// TIA Portal project "SFC_Sep_Simples" (V16)

(* hardware
DEVICE "S71500/ET200MP station_1"  S7-1500 station
   slot 0: "Rail_0"  Rack  6ES7 590-1***0-0AA0
   slot 1: "PLC_1"  CPU 1512C-1 PN  6ES7 512-1CK00-0AB0  V2.8
      slot 3: "CPU display_1"  6ES7591-1AA00-0AA0
      slot 32768: "PROFINET interface_1"  X1
         slot 32769: "Port_1"  X1 P1
         slot 32770: "Port_2"  X1 P2
      slot 34817: "Virtual CP interface port_1"  Virtual CP interface port  Virtual CP interface port
*)

// ===== PLC "PLC_1"  CPU 1512C-1 PN =====

VAR_GLOBAL   // PLC tag table "Default tag table"
   "Count" AT %MW0 : Int;
END_VAR

VAR_GLOBAL   // PLC tag table "E_N_Controlaveis"
   "FIO_S3" AT %M5.3 : Bool;
   "FIO_S2" AT %M5.2 : Bool;
   "FIO_PA" AT %M5.1 : Bool;
   "FIO_PV" AT %M5.0 : Bool;
   "FIO_S4" AT %M5.5 : Bool;
   "FIO_AT_Fwd" AT %M5.6 : Bool;
   "FIOAT_Rev" AT %M5.7 : Bool;
END_VAR

VAR_GLOBAL   // PLC tag table "Saidas"
   "FIO_Atuador" AT %M10.0 : Bool;
   "FIO_Esteira1" AT %M10.1 : Bool;
   "FIO_Esteira2" AT %M10.2 : Bool;
   "FIO_Esteira4" AT %M10.4 : Bool;
   "FIO_Esteira3" AT %M10.3 : Bool;
END_VAR

// folder: DBs

DATA_BLOCK "Eventos"   // DB1
{ S7_Optimized_Access := 'TRUE' }
VERSION : 0.1
   VAR
      PV_Ev : Bool;
      PA_Ev : Bool;
      S2_On_Ev : Bool;
      S2_Off_Ev : Bool;
      S3_On_Ev : Bool;
      S3_Off_Ev : Bool;
      AT_Off_Ev : Bool;
      S4_Off_Ev : Bool;
      AT_On_Ev : Bool;
      E1_On_Ev : Bool;
      E1_Off_Ev : Bool;
      E2_On_Ev : Bool;
      E2_Off_Ev : Bool;
      E3_On_Ev : Bool;
      E3_Off_Ev : Bool;
   END_VAR
BEGIN
END_DATA_BLOCK

DATA_BLOCK "BitsAuxiliares"   // DB2
{ S7_Optimized_Access := 'TRUE' }
VERSION : 0.1
   VAR
      Aux1 : Bool;
      Aux2 : Bool;
      Cont : Int := 0;
   END_VAR
BEGIN
END_DATA_BLOCK

DATA_BLOCK "Sequencia_DB"   // DB6
{ S7_Optimized_Access := 'TRUE' }
VERSION : 0.1
// stored: InstanceOfName Sequencia
"Sequencia"
BEGIN
END_DATA_BLOCK

// folder: System blocks/Program resources

DATA_BLOCK "CT1"   // DB4
{ S7_Optimized_Access := 'TRUE' }
AUTHOR : Simatic
FAMILY : IEC
NAME : CNTR
VERSION : 1.0
// stored: InstanceOfName IEC_COUNTER
"IEC_COUNTER"
BEGIN
END_DATA_BLOCK

// folder: (top level)

ORGANIZATION_BLOCK "Main"   // OB1, LAD, ProgramCycle
TITLE = "Main Program Sweep (Cycle)"
{ S7_Optimized_Access := 'TRUE' }
VERSION : 0.1
   VAR_INPUT
      Initial_Call : Bool;   // Initial call of this OB
      Remanence : Bool;   // =True, if remanent data are available
   END_VAR
   VAR_TEMP   // added for the SCL form of the ladder/FBD networks
      _w1 : Bool;
      _w2 : Bool;
   END_VAR
BEGIN

REGION Network 1: Leituras De Borda
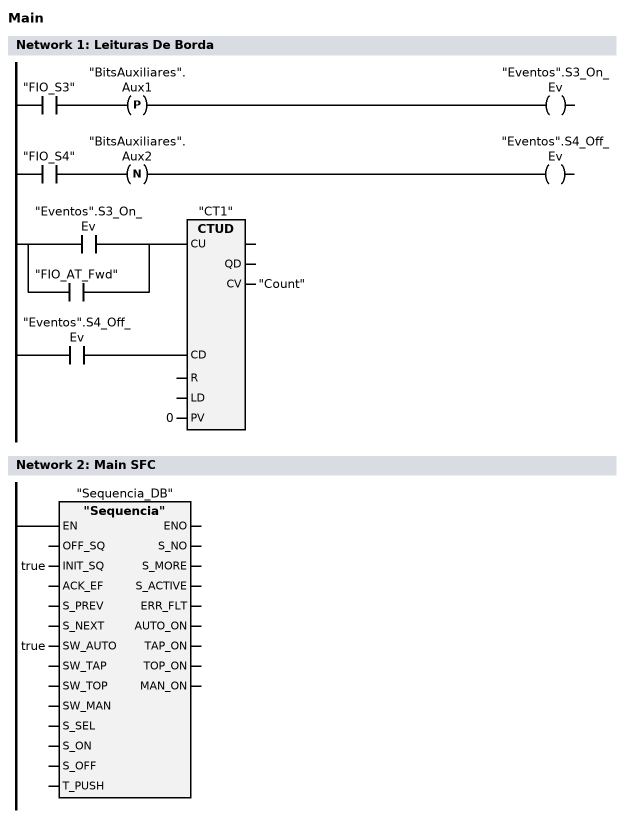
   #_w1 := "FIO_S3" AND NOT "BitsAuxiliares".Aux1;   // rising edge
   "BitsAuxiliares".Aux1 := "FIO_S3";
   "Eventos".S3_On_Ev := #_w1;
   #_w2 := NOT "FIO_S4" AND "BitsAuxiliares".Aux2;   // falling edge
   "BitsAuxiliares".Aux2 := "FIO_S4";
   "Eventos".S4_Off_Ev := #_w2;
   "CT1".CTUD(CU := "Eventos".S3_On_Ev OR "FIO_AT_Fwd", CD := "Eventos".S4_Off_Ev, PV := 0, CV => "Count");
END_REGION

REGION Network 2: Main SFC
   RUNG wire#powerrail
      "Sequencia_DB"(OFF_SQ :=, INIT_SQ := true, ACK_EF :=, S_PREV :=, S_NEXT :=, SW_AUTO := true, SW_TAP :=, SW_TOP :=, SW_MAN :=, S_SEL :=, S_ON :=, S_OFF :=, T_PUSH :=, S_NO =>, S_MORE =>, S_ACTIVE =>, ERR_FLT =>, AUTO_ON =>, TAP_ON =>, TOP_ON =>, MAN_ON =>)
   END_RUNG
   // the same network as SCL:
   "Sequencia_DB"(INIT_SQ := true, SW_AUTO := true);   // "Sequencia"
END_REGION
END_ORGANIZATION_BLOCK

// folder: FBs

FUNCTION_BLOCK "Sequencia"   // FB2, GRAPH_PLUS
{ S7_Optimized_Access := 'TRUE' }
VERSION : 0.1
   VAR_INPUT
      OFF_SQ : Bool := false;   // Turn sequence off
      INIT_SQ : Bool := false;   // Set sequence to initial state
      ACK_EF : Bool := false;   // Acknowledge all errors and faults
      S_PREV : Bool := false;   // Output previous step in parameter S_NO
      S_NEXT : Bool := false;   // Indicate next step in parameter S_NO
      SW_AUTO : Bool := false;   // Automatic mode
      SW_TAP : Bool := false;   // Semiautomatic/switch with transition
      SW_TOP : Bool := false;   // Semiautomatic/ignore transition
      SW_MAN : Bool := false;   // Manual mode
      S_SEL : Int := 0;   // Select step to be output to S_NO
      S_ON : Bool := false;   // Activate step indicated in S_NO
      S_OFF : Bool := false;   // Deactivate step indicated S_NO
      T_PUSH : Bool := false;   // Enable transition to switch in semi automatic mode
   END_VAR
   VAR_OUTPUT
      S_NO : Int := 0;   // Step number
      S_MORE : Bool := false;   // More steps are available and can be shown in S_NO
      S_ACTIVE : Bool := false;   // Step indicated in S_NO is active
      ERR_FLT : Bool := false;   // Interlock or supervision group error
      AUTO_ON : Bool := false;   // Automatic mode is active
      TAP_ON : Bool := false;   // Semiautomatic mode/step with transition enabled
      TOP_ON : Bool := false;   // Semiautomatic mode/ignore transition enabled
      MAN_ON : Bool := false;   // Manual mode is active
   END_VAR
   VAR
      HMI_INFO : Array[0..8] of UInt;
      IF_PAR : G7_IfParPlus_V6;
      RT_DATA : G7_RTDataPlus_V6;   // Internal data area
      Trans1 : G7_TransitionPlus_V6;   // Transition structure
      Trans2 : G7_TransitionPlus_V6;   // Transition structure
      Trans3 : G7_TransitionPlus_V6;   // Transition structure
      Trans4 : G7_TransitionPlus_V6;   // Transition structure
      Trans5 : G7_TransitionPlus_V6;   // Transition structure
      Trans6 : G7_TransitionPlus_V6;   // Transition structure
      Trans7 : G7_TransitionPlus_V6;   // Transition structure
      Trans8 : G7_TransitionPlus_V6;   // Transition structure
      Trans10 : G7_TransitionPlus_V6;   // Transition structure
      Trans12 : G7_TransitionPlus_V6;   // Transition structure
      Trans13 : G7_TransitionPlus_V6;   // Transition structure
      Trans14 : G7_TransitionPlus_V6;   // Transition structure
      Trans15 : G7_TransitionPlus_V6;   // Transition structure
      Trans16 : G7_TransitionPlus_V6;   // Transition structure
      Trans17 : G7_TransitionPlus_V6;   // Transition structure
      Step1 : G7_StepPlus_V6;   // Step structure
      Step2 : G7_StepPlus_V6;   // Step structure
      Step3 : G7_StepPlus_V6;   // Step structure
      Step4 : G7_StepPlus_V6;   // Step structure
      Step5 : G7_StepPlus_V6;   // Step structure
      Step6 : G7_StepPlus_V6;   // Step structure
      Step7 : G7_StepPlus_V6;   // Step structure
      Step9 : G7_StepPlus_V6;   // Step structure
      Step11 : G7_StepPlus_V6;   // Step structure
      Step12 : G7_StepPlus_V6;   // Step structure
      Step13 : G7_StepPlus_V6;   // Step structure
      SINI : Array[0..1] of USInt;
      LSTT : Array[0..14] of USInt;
      ATAJ : Array[0..14] of USInt;
      ATAB : Array[0..14] of USInt;
      PSTT : Array[0..14] of USInt;
      NSTT : Array[0..14] of USInt;
      ASSJ : Array[0..10] of USInt;
      ASSB : Array[0..10] of USInt;
      PTTS : Array[0..10] of USInt;
      NTTS : Array[0..10] of USInt;
      SW_SQTS : Array[0..10] of USInt;
      SWITCH : Array[0..3] of USInt;
      TVX : Array[0..7] of USInt;
      TTX : Array[0..7] of USInt;
      TSX : Array[0..1] of USInt;
      S00X : Array[0..1] of USInt;
      SOFFX : Array[0..1] of USInt;
      SONX : Array[0..1] of USInt;
      SAX : Array[0..1] of USInt;
      SERRX : Array[0..11] of USInt;
      SMX : Array[0..11] of USInt;
      S0X : Array[0..11] of USInt;
      S1X : Array[0..11] of USInt;
      IL_ALARM_INST : Diag_Alarm;
      SUP_ALARM_INST : Diag_Alarm;
      STEP_TIME_ALARM_INST : Diag_Alarm;
      IEC_TIMER_INST : IEC_TIMER;
      TRANSACTION_FLAG : Bool := false;
   END_VAR
   // SINI[0] := 2;
   // LSTT[0] := 255;
   // LSTT[1] := 255;
   // LSTT[2] := 255;
   // LSTT[3] := 255;
   // LSTT[4] := 255;
   // LSTT[5] := 255;
   // LSTT[6] := 255;
   // LSTT[7] := 255;
   // LSTT[8] := 4;
   // LSTT[9] := 255;
   // LSTT[11] := 5;
   // LSTT[12] := 7;
   // LSTT[13] := 255;
   // LSTT[14] := 8;
   // ATAJ[1] := 1;
   // ATAJ[2] := 2;
   // ATAJ[3] := 3;
   // ATAJ[4] := 4;
   // ATAJ[5] := 5;
   // ATAJ[6] := 6;
   // ATAJ[7] := 7;
   // ATAJ[8] := 8;
   // ATAJ[9] := 9;
   // ATAJ[10] := 10;
   // ATAJ[11] := 11;
   // ATAJ[12] := 12;
   // ATAJ[13] := 13;
   // ATAJ[14] := 14;
   // ATAB[1] := 1;
   // ATAB[2] := 2;
   // ATAB[3] := 12;
   // ATAB[4] := 3;
   // ATAB[5] := 5;
   // ATAB[6] := 7;
   // ATAB[7] := 6;
   // ATAB[8] := 8;
   // ATAB[9] := 9;
   // ATAB[10] := 10;
   // ATAB[11] := 4;
   // ATAB[12] := 11;
   // ATAB[13] := 13;
   // ATAB[14] := 14;
   // PSTT[1] := 1;
   // PSTT[2] := 2;
   // PSTT[3] := 3;
   // PSTT[4] := 3;
   // PSTT[5] := 4;
   // PSTT[6] := 10;
   // PSTT[7] := 10;
   // PSTT[8] := 7;
   // PSTT[9] := 8;
   // PSTT[10] := 9;
   // PSTT[11] := 3;
   // PSTT[12] := 3;
   // PSTT[13] := 5;
   // PSTT[14] := 6;
   // NSTT[0] := 1;
   // NSTT[1] := 2;
   // NSTT[2] := 3;
   // NSTT[3] := 8;
   // NSTT[4] := 4;
   // NSTT[5] := 5;
   // NSTT[6] := 6;
   // NSTT[7] := 7;
   // NSTT[8] := 4;
   // NSTT[9] := 9;
   // NSTT[11] := 5;
   // NSTT[12] := 7;
   // NSTT[13] := 10;
   // NSTT[14] := 8;
   // ASSJ[1] := 1;
   // ASSJ[2] := 2;
   // ASSJ[3] := 3;
   // ASSJ[4] := 4;
   // ASSJ[5] := 5;
   // ASSJ[6] := 6;
   // ASSJ[7] := 7;
   // ASSJ[8] := 8;
   // ASSJ[9] := 9;
   // ASSJ[10] := 10;
   // ASSB[1] := 1;
   // ASSB[2] := 2;
   // ASSB[3] := 3;
   // ASSB[4] := 4;
   // ASSB[5] := 5;
   // ASSB[6] := 6;
   // ASSB[7] := 7;
   // ASSB[8] := 8;
   // ASSB[9] := 9;
   // ASSB[10] := 10;
   // PTTS[0] := 255;
   // PTTS[2] := 1;
   // PTTS[3] := 2;
   // PTTS[4] := 4;
   // PTTS[5] := 5;
   // PTTS[6] := 6;
   // PTTS[7] := 7;
   // PTTS[8] := 3;
   // PTTS[9] := 9;
   // PTTS[10] := 13;
   // NTTS[1] := 1;
   // NTTS[2] := 2;
   // NTTS[3] := 3;
   // NTTS[4] := 5;
   // NTTS[5] := 13;
   // NTTS[6] := 14;
   // NTTS[7] := 8;
   // NTTS[8] := 9;
   // NTTS[9] := 10;
   // NTTS[10] := 6;
   // SW_SQTS[4] := 1;
   // SW_SQTS[5] := 1;
   // SW_SQTS[6] := 2;
   // SW_SQTS[7] := 3;
   // SW_SQTS[8] := 4;
   // SW_SQTS[9] := 4;
   // SW_SQTS[10] := 1;
   // TVX[0] := 16#1;
   // TTX[0] := 16#1;
   // TSX[0] := 16#1;
   // S00X[0] := 16#1;
   // SOFFX[0] := 16#1;
   // SONX[0] := 16#1;
   // SAX[0] := 16#1;
   // SERRX[0] := 16#1;
   // SMX[0] := 16#1;
   // S0X[0] := 16#1;
   // S1X[0] := 16#1;
BEGIN
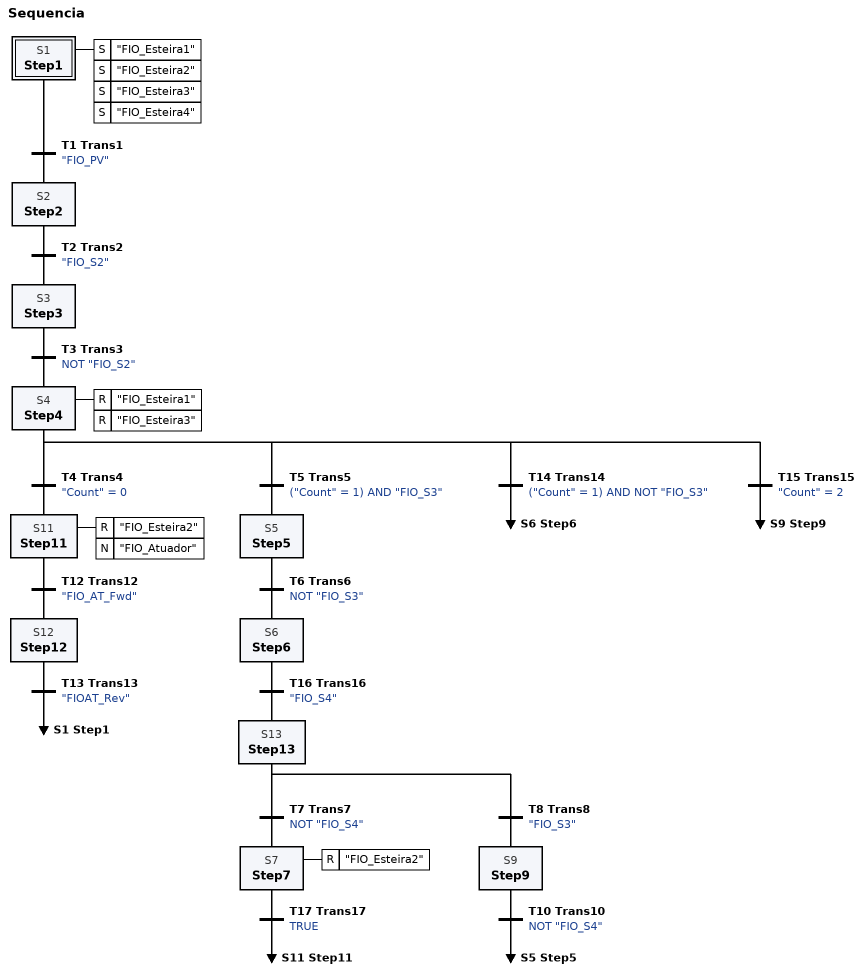
   // sequencer 1
   INITIAL_STEP Step1:   // S1, max time T#10S, warning time T#7S
              S    "FIO_Esteira1"
              S    "FIO_Esteira2"
              S    "FIO_Esteira3"
              S    "FIO_Esteira4"
   END_STEP
   TRANSITION Trans1 FROM Step1 TO Step2   // T1
      := "FIO_PV";
   END_TRANSITION
   STEP Step2:   // S2, max time T#10S, warning time T#7S
   END_STEP
   TRANSITION Trans2 FROM Step2 TO Step3   // T2
      := "FIO_S2";
   END_TRANSITION
   STEP Step3:   // S3, max time T#10S, warning time T#7S
   END_STEP
   TRANSITION Trans3 FROM Step3 TO Step4   // T3
      := NOT "FIO_S2";
   END_TRANSITION
   STEP Step4:   // S4, max time T#10S, warning time T#7S
              R    "FIO_Esteira1"
              R    "FIO_Esteira3"
   END_STEP
   TRANSITION Trans4 FROM Step4 TO Step11   // T4
      := "Count" = 0;
   END_TRANSITION
   TRANSITION Trans5 FROM Step4 TO Step5   // T5
      := ("Count" = 1) AND "FIO_S3";
   END_TRANSITION
   TRANSITION Trans14 FROM Step4 TO Step6   // T14, jump
      := ("Count" = 1) AND NOT "FIO_S3";
   END_TRANSITION
   TRANSITION Trans15 FROM Step4 TO Step9   // T15, jump
      := "Count" = 2;
   END_TRANSITION
   STEP Step5:   // S5, max time T#10S, warning time T#7S
   END_STEP
   TRANSITION Trans6 FROM Step5 TO Step6   // T6
      := NOT "FIO_S3";
   END_TRANSITION
   STEP Step6:   // S6, max time T#10S, warning time T#7S
   END_STEP
   TRANSITION Trans16 FROM Step6 TO Step13   // T16
      := "FIO_S4";
   END_TRANSITION
   STEP Step7:   // S7, max time T#10S, warning time T#7S
              R    "FIO_Esteira2"
   END_STEP
   TRANSITION Trans17 FROM Step7 TO Step11   // T17, jump
      := TRUE;
   END_TRANSITION
   STEP Step9:   // S9, max time T#10S, warning time T#7S
   END_STEP
   TRANSITION Trans10 FROM Step9 TO Step5   // T10, jump
      := NOT "FIO_S4";
   END_TRANSITION
   STEP Step11:   // S11, max time T#10S, warning time T#7S
              R    "FIO_Esteira2"
              N    "FIO_Atuador"
   END_STEP
   TRANSITION Trans12 FROM Step11 TO Step12   // T12
      := "FIO_AT_Fwd";
   END_TRANSITION
   STEP Step12:   // S12, max time T#10S, warning time T#7S
   END_STEP
   TRANSITION Trans13 FROM Step12 TO Step1   // T13, jump
      := "FIOAT_Rev";
   END_TRANSITION
   STEP Step13:   // S13, max time T#10S, warning time T#7S
   END_STEP
   TRANSITION Trans7 FROM Step13 TO Step7   // T7
      := NOT "FIO_S4";
   END_TRANSITION
   TRANSITION Trans8 FROM Step13 TO Step9   // T8
      := "FIO_S3";
   END_TRANSITION
END_FUNCTION_BLOCK